FUNCTION_BLOCK CommFromMatlab3 (* Extracted Composite Function Block Type *)
  (* Version 5/20/2016, gulzha *)
  PACKAGE Main;
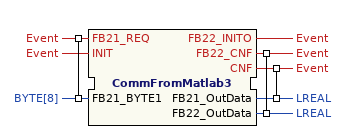
  EVENT_INPUT
    FB21_REQ WITH FB21_BYTE1; (* Normal Execution Request *)
    INIT; (* Initialization Request *)
  END_EVENT
  EVENT_OUTPUT
    FB22_INITO; (* Initialization Confirm *)
    FB22_CNF WITH FB22_OutData; (* Execution Confirmation *)
    CNF WITH FB21_OutData; (* Execution Confirmation *)
  END_EVENT
  VAR_INPUT
    FB21_BYTE1 : ARRAY [0..7] OF BYTE;
  END_VAR
  VAR_OUTPUT
    FB21_OutData : LREAL;
    FB22_OutData : LREAL;
  END_VAR
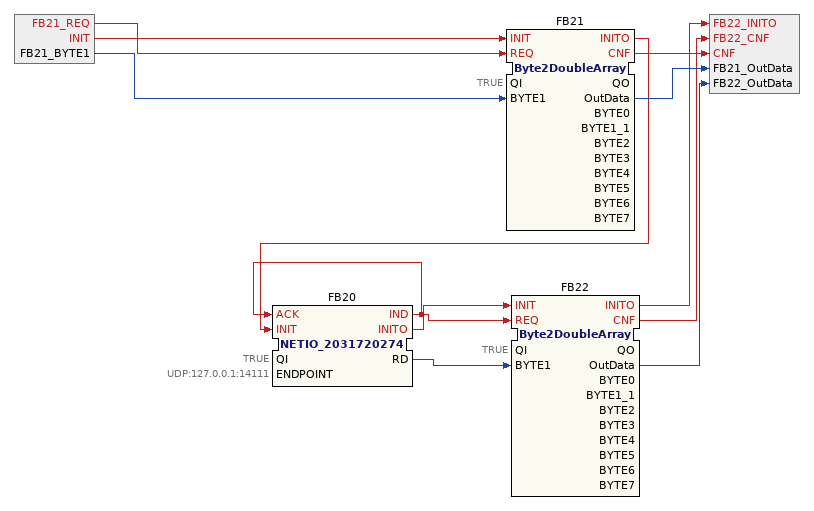
  FBS
    FB20 : NETIO_2031720274(QI := TRUE, ENDPOINT := UDP:127.0.0.1:14111); {SET_ATTRIBUTE(Configuration.GenericFBType.InterfaceParams, Runtime.IoCommon#I:=1;SD:BYTE[8];RD:BYTE[8])}
    FB21 : Byte2DoubleArray(QI := TRUE);
    FB22 : Byte2DoubleArray(QI := TRUE);
  END_FBS
  EVENT_CONNECTIONS
    FB20.IND TO FB20.ACK;
    FB21.INITO TO FB20.INIT;
    FB20.INITO TO FB22.INIT;
    FB20.IND TO FB22.REQ;
    FB21_REQ TO FB21.REQ;
    FB22.INITO TO FB22_INITO;
    FB22.CNF TO FB22_CNF;
    FB21.CNF TO CNF;
    INIT TO FB21.INIT;
  END_CONNECTIONS
  DATA_CONNECTIONS
    FB20.RD TO FB22.BYTE1;
    FB21_BYTE1 TO FB21.BYTE1;
    FB21.OutData TO FB21_OutData;
    FB22.OutData TO FB22_OutData;
  END_CONNECTIONS
END_FUNCTION_BLOCK
